// TIA Portal project "Lab04-datalog" (V17)

(* hardware
DEVICE "S7-1200 station_1"  S7-1200 Station
   slot 0: "Rack_0"  S7-1200 Rack  Rack  V1.0
   slot 1: "PLC_1"  CPU 1214C DC/DC/DC  6ES7 214-1AG40-0XB0  V4.4
*)

// ===== PLC "PLC_1"  CPU 1214C DC/DC/DC =====

VAR_GLOBAL   // PLC tag table "Default tag table"
   "Tag_1" AT %M2.0 : Bool;
   "System_Byte" AT %MB1 : Byte;
   "FirstScan" AT %M1.0 : Bool;
   "DiagStatusUpdate" AT %M1.1 : Bool;
   "AlwaysTRUE" AT %M1.2 : Bool;
   "AlwaysFALSE" AT %M1.3 : Bool;
   "Clock_Byte" AT %MB0 : Byte;
   "Clock_10Hz" AT %M0.0 : Bool;
   "Clock_5Hz" AT %M0.1 : Bool;
   "Clock_2.5Hz" AT %M0.2 : Bool;
   "Clock_2Hz" AT %M0.3 : Bool;
   "Clock_1.25Hz" AT %M0.4 : Bool;
   "Clock_1Hz" AT %M0.5 : Bool;
   "Clock_0.625Hz" AT %M0.6 : Bool;
   "Clock_0.5Hz" AT %M0.7 : Bool;
END_VAR

TYPE "UDT_Medidor"
   STRUCT
      Voltaje : Real;
      Corriente : Real;
      Potencia : Real;
   END_STRUCT;
END_TYPE

DATA_BLOCK "Datalog_Vars"   // DB1
{ S7_Optimized_Access := 'TRUE' }
VERSION : 0.1
   VAR
      DataLogName : String := 'MiDataLog';
      DataLogID : DWord := 0;
      DataLogHeaders : String := 'Voltaje,Corriente,Potencial';
      Data : Struct
         Voltaje : Real;
         Corriente : Real;
         Potencia : Real;
      END_STRUCT;
   END_VAR
BEGIN
END_DATA_BLOCK

DATA_BLOCK "Medidores"   // DB2
{ S7_Optimized_Access := 'TRUE' }
VERSION : 0.1
   VAR
      Medidor1 : "UDT_Medidor";
      Medidor2 : "UDT_Medidor";
      Medidor3 : "UDT_Medidor";
      Medidor4 : "UDT_Medidor";
      Medidor5 : "UDT_Medidor";
      Medidor6 : "UDT_Medidor";
      Medidor7 : "UDT_Medidor";
      Medidor8 : "UDT_Medidor";
      Medidor9 : "UDT_Medidor";
      Medidor10 : "UDT_Medidor";
   END_VAR
BEGIN
END_DATA_BLOCK

DATA_BLOCK "FB_DataLog_DB"   // DB3
{ S7_Optimized_Access := 'TRUE' }
VERSION : 0.1
// stored: InstanceOfName FB_DataLog
"FB_DataLog"
BEGIN
END_DATA_BLOCK

FUNCTION_BLOCK "FB_DataLog"   // FB1, LAD
{ S7_Optimized_Access := 'TRUE' }
VERSION : 0.1
   VAR
      DataLogCreate_Instance : DataLogCreate;
      aux1 : Bool;
      DataLogCreated : Bool;
      SaveStatusCreated : Word;
      aux2 : Bool;
      aux3 : Bool;
      aux4 : Bool;
      DataLogWrite_Instance : DataLogWrite;
      DataLogClose_Instance : DataLogClose;
   END_VAR
   VAR_TEMP
      CreateDone : Bool;
      CreateBusy : Bool;
      CreateError : Bool;
      CreateStatus : Word;
      WriteDone : Bool;
      WriteBussy : Bool;
      WriteError : Bool;
      WriteStatus : Word;
   END_VAR
   VAR_TEMP   // added for the SCL form of the ladder/FBD networks
      _w1 : Bool;
   END_VAR
BEGIN

REGION Network 1
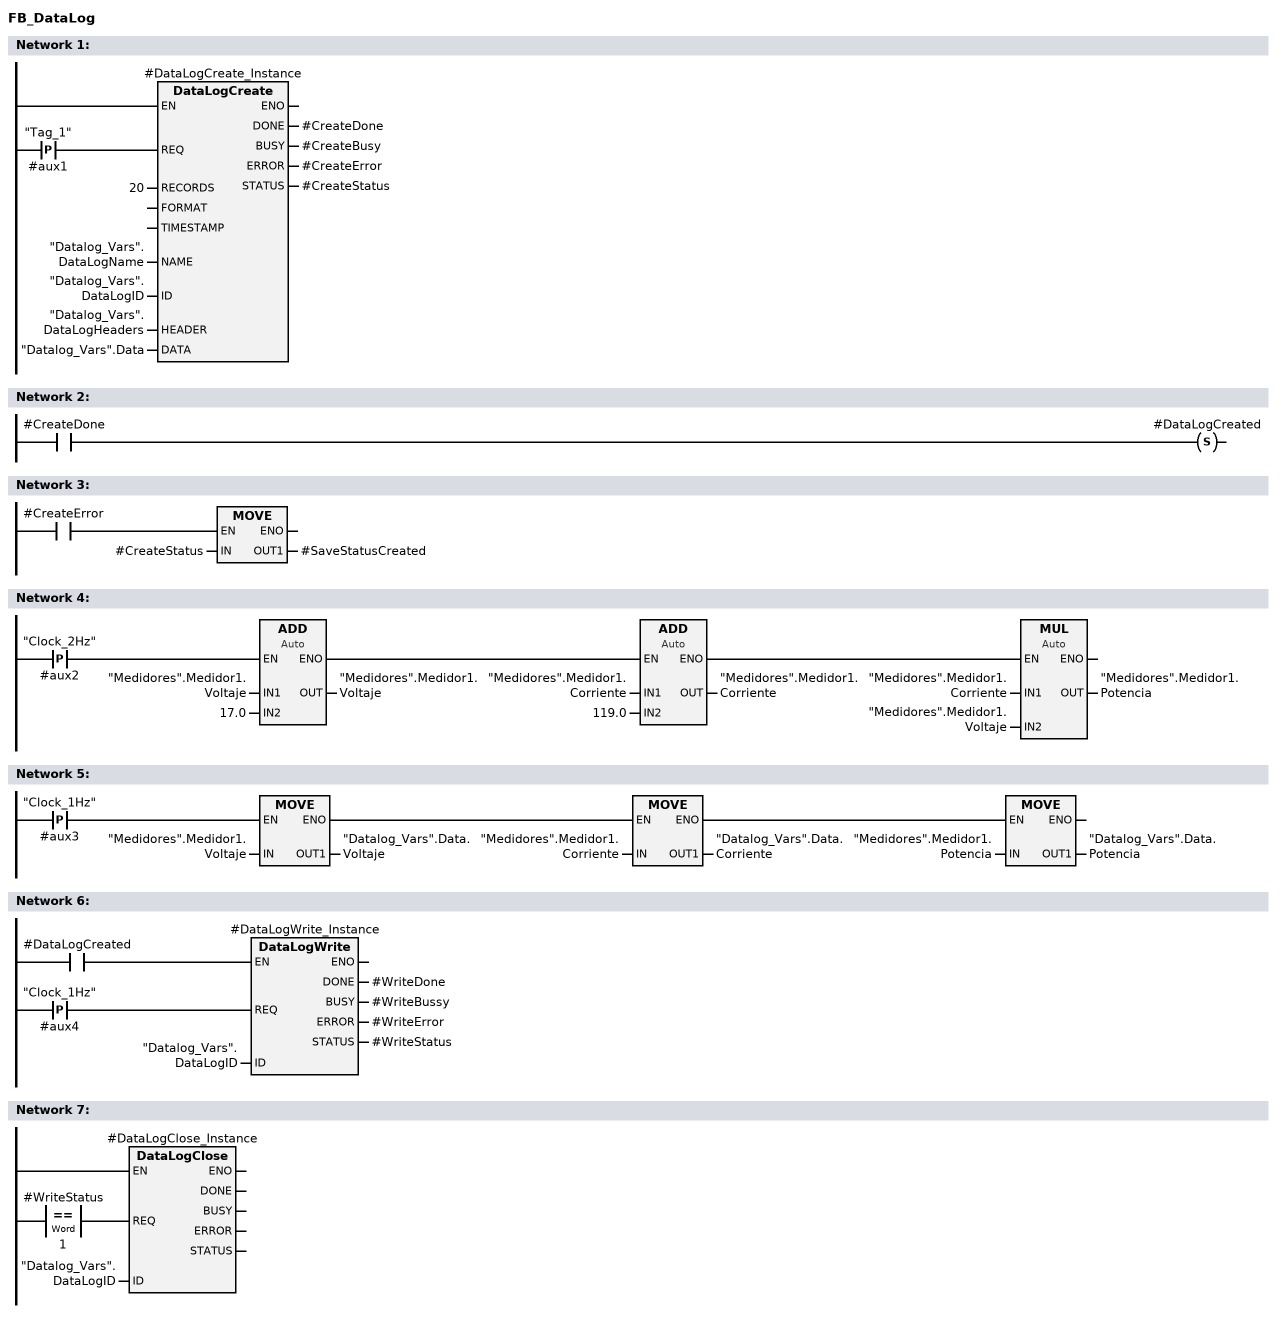
   #_w1 := "Tag_1" AND NOT #aux1;   // rising edge of "Tag_1"
   #aux1 := "Tag_1";
   #DataLogCreate_Instance(REQ := #_w1,   // DataLogCreate
                           RECORDS := 20,
                           "NAME" := "Datalog_Vars".DataLogName,
                           ID := "Datalog_Vars".DataLogID,
                           HEADER := "Datalog_Vars".DataLogHeaders,
                           DATA := "Datalog_Vars".Data,
                           DONE => #CreateDone,
                           BUSY => #CreateBusy,
                           ERROR => #CreateError,
                           STATUS => #CreateStatus);
END_REGION

REGION Network 2
   RUNG wire#powerrail
      Contact( #CreateDone )
      S_Coil( #DataLogCreated )
   END_RUNG
   // the same network as SCL:
   IF #CreateDone THEN #DataLogCreated := TRUE; END_IF;
END_REGION

REGION Network 3
   RUNG wire#powerrail
      Contact( #CreateError )
      Move(in := #CreateStatus, out1 => #SaveStatusCreated)
   END_RUNG
   // the same network as SCL:
   IF #CreateError THEN #SaveStatusCreated := #CreateStatus; END_IF;
END_REGION

REGION Network 4
   RUNG wire#powerrail
      P_Contact(operand := "Clock_2Hz", bit := #aux2)
      Add(in1 := "Medidores".Medidor1.Voltaje, in2 := 17.0, out => "Medidores".Medidor1.Voltaje)
      Add(in1 := "Medidores".Medidor1.Corriente, in2 := 119.0, out => "Medidores".Medidor1.Corriente)
      Mul(in1 := "Medidores".Medidor1.Corriente, in2 := "Medidores".Medidor1.Voltaje, out => "Medidores".Medidor1.Potencia)
   END_RUNG
   // the same network as SCL:
   #_w1 := "Clock_2Hz" AND NOT #aux2;   // rising edge of "Clock_2Hz"
   #aux2 := "Clock_2Hz";
   IF #_w1 THEN
       "Medidores".Medidor1.Voltaje := "Medidores".Medidor1.Voltaje + 17.0;
       "Medidores".Medidor1.Corriente := "Medidores".Medidor1.Corriente + 119.0;
       "Medidores".Medidor1.Potencia := "Medidores".Medidor1.Corriente * "Medidores".Medidor1.Voltaje;
   END_IF;
END_REGION

REGION Network 5
   RUNG wire#powerrail
      P_Contact(operand := "Clock_1Hz", bit := #aux3)
      Move(in := "Medidores".Medidor1.Voltaje, out1 => "Datalog_Vars".Data.Voltaje)
      Move(in := "Medidores".Medidor1.Corriente, out1 => "Datalog_Vars".Data.Corriente)
      Move(in := "Medidores".Medidor1.Potencia, out1 => "Datalog_Vars".Data.Potencia)
   END_RUNG
   // the same network as SCL:
   #_w1 := "Clock_1Hz" AND NOT #aux3;   // rising edge of "Clock_1Hz"
   #aux3 := "Clock_1Hz";
   IF #_w1 THEN
       "Datalog_Vars".Data.Voltaje := "Medidores".Medidor1.Voltaje;
       "Datalog_Vars".Data.Corriente := "Medidores".Medidor1.Corriente;
       "Datalog_Vars".Data.Potencia := "Medidores".Medidor1.Potencia;
   END_IF;
END_REGION

REGION Network 6
   #_w1 := "Clock_1Hz" AND NOT #aux4;   // rising edge of "Clock_1Hz"
   #aux4 := "Clock_1Hz";
   IF #DataLogCreated THEN
       #DataLogWrite_Instance(REQ := #_w1,   // DataLogWrite
                              ID := "Datalog_Vars".DataLogID,
                              DONE => #WriteDone,
                              BUSY => #WriteBussy,
                              ERROR => #WriteError,
                              STATUS => #WriteStatus);
   END_IF;
END_REGION

REGION Network 7
   #DataLogClose_Instance(REQ := #WriteStatus = 1, ID := "Datalog_Vars".DataLogID);   // DataLogClose
END_REGION
END_FUNCTION_BLOCK

ORGANIZATION_BLOCK "Main"   // OB1, LAD, ProgramCycle
TITLE = "Main Program Sweep (Cycle)"
{ S7_Optimized_Access := 'TRUE' }
VERSION : 0.1
   VAR_INPUT
      Initial_Call : Bool;   // Initial call of this OB
      Remanence : Bool;   // =True, if remanent data are available
   END_VAR
BEGIN

REGION Network 1
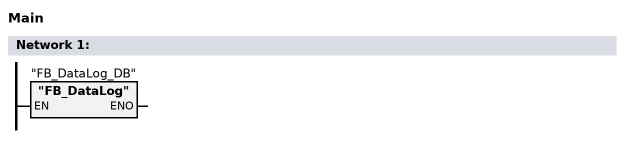
   RUNG wire#powerrail
      "FB_DataLog_DB"()
   END_RUNG
   // the same network as SCL:
   "FB_DataLog_DB"();   // "FB_DataLog"
END_REGION
END_ORGANIZATION_BLOCK